// TIA Portal project "Liquid_Level_Control_Factory_IO" (V15)
// Vorlageprojekt für das Buch mit Zielsystem S7-1200

(* hardware
DEVICE "S7-1200-Station_1"  S7-1200 Station
   slot 0: "Baugruppenträger_0"  Rack  V1.0
   slot 1: "Liquid_Level_PLC"  CPU 1211C DC/DC/DC  6ES7 211-1AE40-0XB0  V4.1
DEVICE "Liquid_Level_HMI"  KTP900 Basic PN
   slot 0: "Liquid_Level_HMI"  KTP900 Basic PN  6AV2 123-2JB03-0AX0  15.0.0.0
   slot 1: "HMI_RT_1"  KTP900 Basic PN  6AV2 123-2JB03-0AX0  15.0.0.0
   slot 5: "Liquid_Level_HMI.IE_CP_1"  PROFINET Interface  15.0.0.0
      slot 1: "PROFINET Interface_1"  PROFINET Interface
         slot 1: "Port_1"  Port
*)

// ===== PLC "Liquid_Level_PLC"  CPU 1211C DC/DC/DC =====

VAR_GLOBAL   // PLC tag table "Standard-Variablentabelle"
   "SETPOINT_BUFF" AT %MD100 : DWord;
   "LEVEL_METER_BUFF" AT %MD108 : Real;
   "Discharge_Valve_Buff" AT %MD116 : Real;
END_VAR

VAR_GLOBAL   // PLC tag table "Actuators"
   "START_LGT" AT %Q0.0 : Bool;
   "RESET_LGT" AT %Q0.1 : Bool;
   "STOP_LGT" AT %Q0.2 : Bool;
   "FILL_VALVE" AT %QW30 : Int;
   "DISCHARGE_VALVE" AT %QW32 : Int;
   "WARNING_LGT" AT %Q0.3 : Bool;
   "SIREN" AT %Q0.4 : Bool;
END_VAR

VAR_GLOBAL   // PLC tag table "Sensors"
   "LEVEL_METER" AT %IW30 : Int;
   "FLOW_METER" AT %IW32 : Int;
   "SETPOINT" AT %IW34 : Int;
END_VAR

VAR_GLOBAL   // PLC tag table "Buttons"
   "START_BTN" AT %I0.0 : Bool;
   "RESET_BTN" AT %I0.1 : Bool;
   "STOP_BTN" AT %I0.2 : Bool;
END_VAR

VAR_GLOBAL   // PLC tag table "Display"
   "SP" AT %QW34 : Int;
   "PV" AT %QW36 : Int;
END_VAR

DATA_BLOCK "TANK_CTRL_DB_1"   // DB1
{ S7_Optimized_Access := 'TRUE' }
VERSION : 0.1
   VAR
      PV : Int;
      SP : Int;
      Tank_Lvl : Int;
      Fill_Valve_Pos : Real;
      Valve_Animation : Bool;
      Discharge_Valve : Real;
      Discharge_Animation : Bool;
      In_Error : Int;
      Out_Error : Int;
      Sensor_Error : Int;
      SP_Error : Int;
      Discharge_Error : Int;
      PID_Auto_Bit : Bool;
      PID_Calc_Bit : Bool;
      PID_Mode : Struct
         Enable : Int := 3;
         Disable : Int := 0;
      END_STRUCT;
      PID_Parameters : Struct
         Kp : Real;
         Ti : Real;
         Td : Real;
      END_STRUCT;
      Tuning_Parameters : Struct
         Kp : Real := 2.5;
         Ti : Real := 0.0;
         Td : Real := 0.0;
         Kp_D : Real := 2.5;
         Ti_D : Real := 10.0;
         Td_D : Real := 0.0;
      END_STRUCT;
   END_VAR
   VAR RETAIN
      Calc_Parameters : Struct
         Kp : Real := 2.0;
         Ti : Real := 1.7655;
         Td : Real := 0.0;
      END_STRUCT;
   END_VAR
BEGIN
END_DATA_BLOCK

FUNCTION "Tank_Ctrl" : Void   // FC1, LAD
{ S7_Optimized_Access := 'TRUE' }
VERSION : 0.1
BEGIN

REGION Network 1: SCALE SP
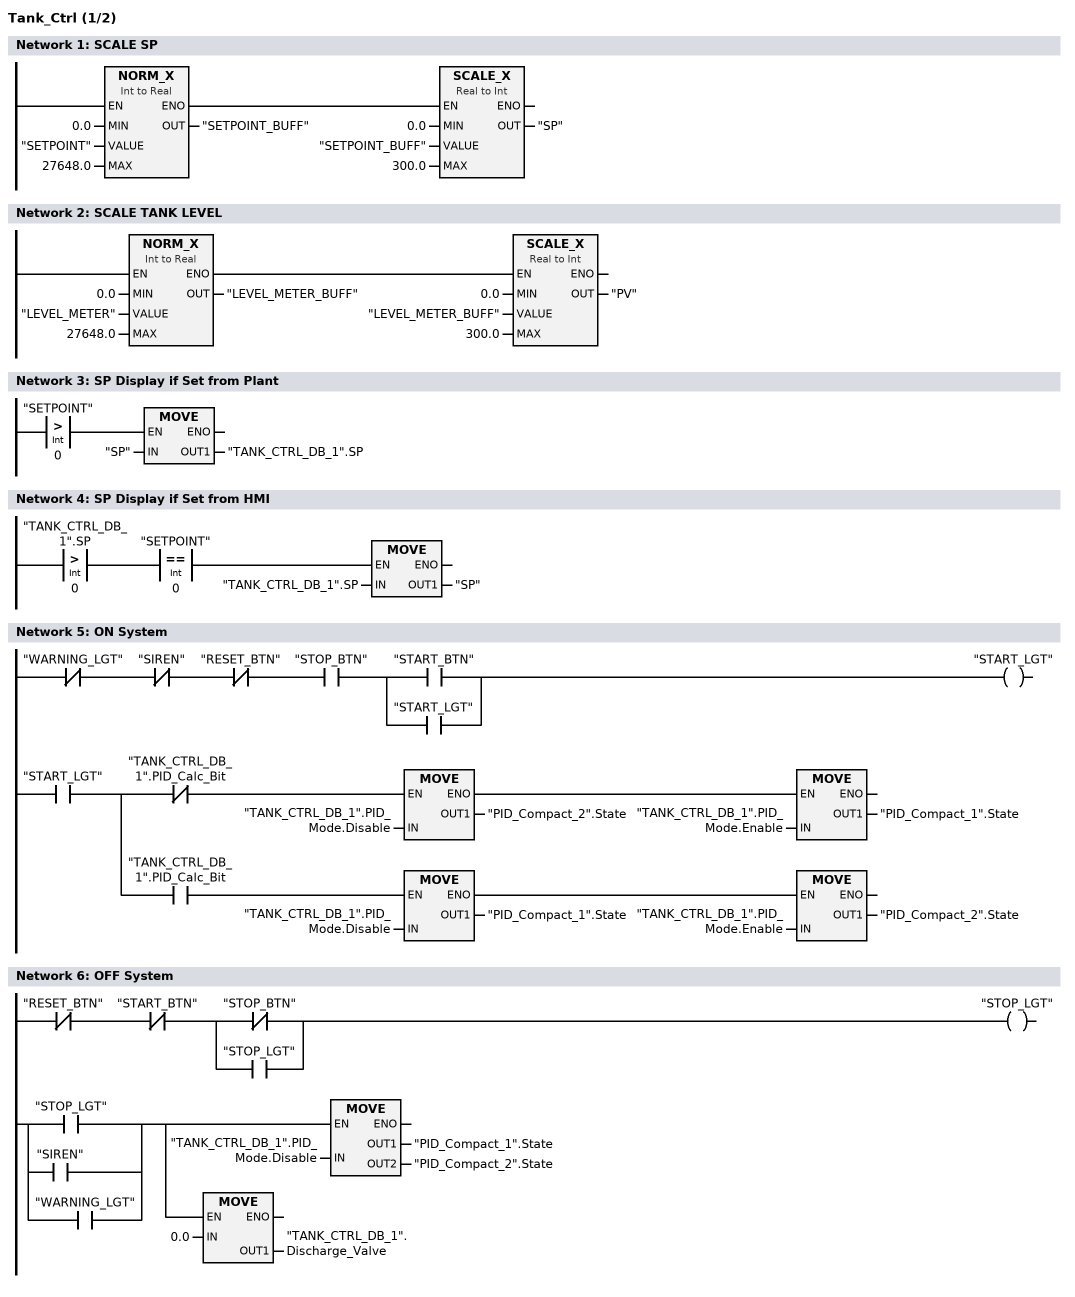
   RUNG wire#powerrail
      { S7_Templates := "[SrcType := Int, DestType := Real]" } Normalize(min := 0.0, value := "SETPOINT", max := 27648.0, out => "SETPOINT_BUFF")
      { S7_Templates := "[SrcType := Real, DestType := Int]" } Scale(min := 0.0, value := "SETPOINT_BUFF", max := 300.0, out => "SP")
   END_RUNG
   // the same network as SCL:
   "SETPOINT_BUFF" := NORM_X(MIN := 0.0, VALUE := "SETPOINT", MAX := 27648.0);
   "SP" := SCALE_X(MIN := 0.0, VALUE := "SETPOINT_BUFF", MAX := 300.0);
END_REGION

REGION Network 2: SCALE TANK LEVEL
   RUNG wire#powerrail
      { S7_Templates := "[SrcType := Int, DestType := Real]" } Normalize(min := 0.0, value := "LEVEL_METER", max := 27648.0, out => "LEVEL_METER_BUFF")
      { S7_Templates := "[SrcType := Real, DestType := Int]" } Scale(min := 0.0, value := "LEVEL_METER_BUFF", max := 300.0, out => "PV")
   END_RUNG
   // the same network as SCL:
   "LEVEL_METER_BUFF" := NORM_X(MIN := 0.0, VALUE := "LEVEL_METER", MAX := 27648.0);
   "PV" := SCALE_X(MIN := 0.0, VALUE := "LEVEL_METER_BUFF", MAX := 300.0);
END_REGION

REGION Network 3: SP Display if Set from Plant
   RUNG wire#powerrail
      { S7_Templates := "SrcType := Int" } GT_Contact(in1 := "SETPOINT", in2 := 0)
      Move(in := "SP", out1 => "TANK_CTRL_DB_1".SP)
   END_RUNG
   // the same network as SCL:
   IF "SETPOINT" > 0 THEN "TANK_CTRL_DB_1".SP := "SP"; END_IF;
END_REGION

REGION Network 4: SP Display if Set from HMI
   RUNG wire#powerrail
      { S7_Templates := "SrcType := Int" } GT_Contact(in1 := "TANK_CTRL_DB_1".SP, in2 := 0)
      { S7_Templates := "SrcType := Int" } EQ_Contact(in1 := "SETPOINT", in2 := 0)
      Move(in := "TANK_CTRL_DB_1".SP, out1 => "SP")
   END_RUNG
   // the same network as SCL:
   IF ("TANK_CTRL_DB_1".SP > 0) AND ("SETPOINT" = 0) THEN "SP" := "TANK_CTRL_DB_1".SP; END_IF;
END_REGION

REGION Network 5: ON System
   RUNG wire#powerrail
      I_Contact( "WARNING_LGT" )
      I_Contact( "SIREN" )
      I_Contact( "RESET_BTN" )
      Contact( "STOP_BTN" )
      wire#w1
      Contact( "START_BTN" )
      wire#w2
      Coil( "START_LGT" )
   END_RUNG
   RUNG wire#w1
      Contact( "START_LGT" )
   END_RUNG wire#w2
   RUNG wire#powerrail
      Contact( "START_LGT" )
      wire#w3
      I_Contact( "TANK_CTRL_DB_1".PID_Calc_Bit )
      Move(in := "TANK_CTRL_DB_1".PID_Mode.Disable, out1 => "PID_Compact_2".State)
      Move(in := "TANK_CTRL_DB_1".PID_Mode.Enable, out1 => "PID_Compact_1".State)
   END_RUNG
   RUNG wire#w3
      Contact( "TANK_CTRL_DB_1".PID_Calc_Bit )
      Move(in := "TANK_CTRL_DB_1".PID_Mode.Disable, out1 => "PID_Compact_1".State)
      Move(in := "TANK_CTRL_DB_1".PID_Mode.Enable, out1 => "PID_Compact_2".State)
   END_RUNG
   // the same network as SCL:
   "START_LGT" := NOT "WARNING_LGT" AND NOT "SIREN" AND NOT "RESET_BTN" AND "STOP_BTN" AND ("START_BTN" OR "START_LGT");
   IF "START_LGT" AND NOT "TANK_CTRL_DB_1".PID_Calc_Bit THEN
       "PID_Compact_2".State := "TANK_CTRL_DB_1".PID_Mode.Disable;
       "PID_Compact_1".State := "TANK_CTRL_DB_1".PID_Mode.Enable;
   END_IF;
   IF "START_LGT" AND "TANK_CTRL_DB_1".PID_Calc_Bit THEN
       "PID_Compact_1".State := "TANK_CTRL_DB_1".PID_Mode.Disable;
       "PID_Compact_2".State := "TANK_CTRL_DB_1".PID_Mode.Enable;
   END_IF;
END_REGION

REGION Network 6: OFF System
   RUNG wire#powerrail
      I_Contact( "RESET_BTN" )
      I_Contact( "START_BTN" )
      wire#w1
      I_Contact( "STOP_BTN" )
      wire#w2
      Coil( "STOP_LGT" )
   END_RUNG
   RUNG wire#w1
      Contact( "STOP_LGT" )
   END_RUNG wire#w2
   RUNG wire#powerrail
      Contact( "STOP_LGT" )
      wire#w3
      Move(in := "TANK_CTRL_DB_1".PID_Mode.Disable, out1 => "PID_Compact_1".State, out2 => "PID_Compact_2".State)
   END_RUNG
   RUNG wire#powerrail
      Contact( "SIREN" )
   END_RUNG wire#w3
   RUNG wire#powerrail
      Contact( "WARNING_LGT" )
   END_RUNG wire#w3
   RUNG wire#w3
      Move(in := 0.0, out1 => "TANK_CTRL_DB_1".Discharge_Valve)
   END_RUNG
   // the same network as SCL:
   "STOP_LGT" := NOT "RESET_BTN" AND NOT "START_BTN" AND (NOT "STOP_BTN" OR "STOP_LGT");
   IF "STOP_LGT" OR "SIREN" OR "WARNING_LGT" THEN
       "PID_Compact_1".State := "TANK_CTRL_DB_1".PID_Mode.Disable;
       "PID_Compact_2".State := "TANK_CTRL_DB_1".PID_Mode.Disable;
       "TANK_CTRL_DB_1".Discharge_Valve := 0.0;
   END_IF;
END_REGION

REGION Network 7: RESET System
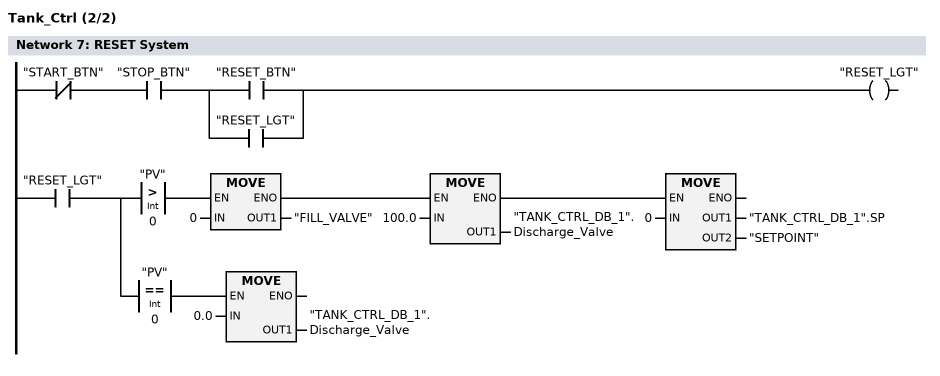
   RUNG wire#powerrail
      I_Contact( "START_BTN" )
      Contact( "STOP_BTN" )
      wire#w1
      Contact( "RESET_BTN" )
      wire#w2
      Coil( "RESET_LGT" )
   END_RUNG
   RUNG wire#w1
      Contact( "RESET_LGT" )
   END_RUNG wire#w2
   RUNG wire#powerrail
      Contact( "RESET_LGT" )
      wire#w3
      { S7_Templates := "SrcType := Int" } GT_Contact(in1 := "PV", in2 := 0)
      Move(in := 0, out1 => "FILL_VALVE")
      Move(in := 100.0, out1 => "TANK_CTRL_DB_1".Discharge_Valve)
      Move(in := 0, out1 => "TANK_CTRL_DB_1".SP, out2 => "SETPOINT")
   END_RUNG
   RUNG wire#w3
      { S7_Templates := "SrcType := Int" } EQ_Contact(in1 := "PV", in2 := 0)
      Move(in := 0.0, out1 => "TANK_CTRL_DB_1".Discharge_Valve)
   END_RUNG
   // the same network as SCL:
   "RESET_LGT" := NOT "START_BTN" AND "STOP_BTN" AND ("RESET_BTN" OR "RESET_LGT");
   IF "RESET_LGT" AND ("PV" > 0) THEN
       "FILL_VALVE" := 0;
       "TANK_CTRL_DB_1".Discharge_Valve := 100.0;
       "TANK_CTRL_DB_1".SP := 0;
       "SETPOINT" := 0;
   END_IF;
   IF "RESET_LGT" AND ("PV" = 0) THEN "TANK_CTRL_DB_1".Discharge_Valve := 0.0; END_IF;
END_REGION
END_FUNCTION

FUNCTION "HMI_Ctrl" : Void   // FC2, LAD
{ S7_Optimized_Access := 'TRUE' }
VERSION : 0.1
   VAR_TEMP   // added for the SCL form of the ladder/FBD networks
      _w1 : Bool;
      _w2 : Bool;
   END_VAR
BEGIN

REGION Network 1: PV and Tank Level
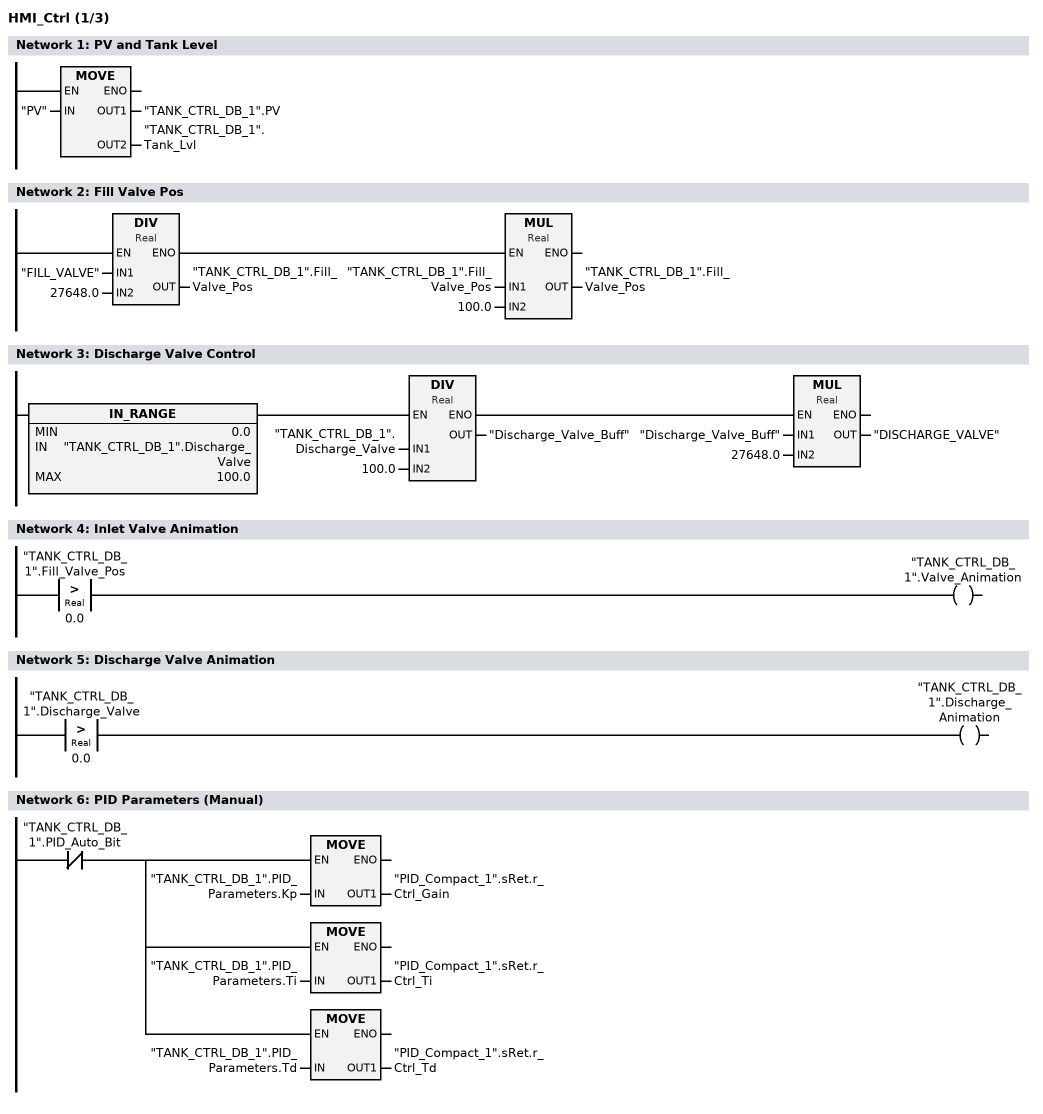
   RUNG wire#powerrail
      Move(in := "PV", out1 => "TANK_CTRL_DB_1".PV, out2 => "TANK_CTRL_DB_1".Tank_Lvl)
   END_RUNG
   // the same network as SCL:
   "TANK_CTRL_DB_1".PV := "PV";
   "TANK_CTRL_DB_1".Tank_Lvl := "PV";
END_REGION

REGION Network 2: Fill Valve Pos
   RUNG wire#powerrail
      { S7_Templates := "SrcType := Real" } Div(in1 := "FILL_VALVE", in2 := 27648.0, out => "TANK_CTRL_DB_1".Fill_Valve_Pos)
      { S7_Templates := "SrcType := Real" } Mul(in1 := "TANK_CTRL_DB_1".Fill_Valve_Pos, in2 := 100.0, out => "TANK_CTRL_DB_1".Fill_Valve_Pos)
   END_RUNG
   // the same network as SCL:
   "TANK_CTRL_DB_1".Fill_Valve_Pos := "FILL_VALVE" / 27648.0;
   "TANK_CTRL_DB_1".Fill_Valve_Pos := "TANK_CTRL_DB_1".Fill_Valve_Pos * 100.0;
END_REGION

REGION Network 3: Discharge Valve Control
   RUNG wire#powerrail
      { S7_Templates := "SrcType := Real" } InRange(min := 0.0, in := "TANK_CTRL_DB_1".Discharge_Valve, max := 100.0)
      { S7_Templates := "SrcType := Real" } Div(in1 := "TANK_CTRL_DB_1".Discharge_Valve, in2 := 100.0, out => "Discharge_Valve_Buff")
      { S7_Templates := "SrcType := Real" } Mul(in1 := "Discharge_Valve_Buff", in2 := 27648.0, out => "DISCHARGE_VALVE")
   END_RUNG
   // the same network as SCL:
   IF (0.0 <= "TANK_CTRL_DB_1".Discharge_Valve) AND ("TANK_CTRL_DB_1".Discharge_Valve <= 100.0) THEN
       "Discharge_Valve_Buff" := "TANK_CTRL_DB_1".Discharge_Valve / 100.0;
       "DISCHARGE_VALVE" := "Discharge_Valve_Buff" * 27648.0;
   END_IF;
END_REGION

REGION Network 4: Inlet Valve Animation
   RUNG wire#powerrail
      { S7_Templates := "SrcType := Real" } GT_Contact(in1 := "TANK_CTRL_DB_1".Fill_Valve_Pos, in2 := 0.0)
      Coil( "TANK_CTRL_DB_1".Valve_Animation )
   END_RUNG
   // the same network as SCL:
   "TANK_CTRL_DB_1".Valve_Animation := "TANK_CTRL_DB_1".Fill_Valve_Pos > 0.0;
END_REGION

REGION Network 5: Discharge Valve Animation
   RUNG wire#powerrail
      { S7_Templates := "SrcType := Real" } GT_Contact(in1 := "TANK_CTRL_DB_1".Discharge_Valve, in2 := 0.0)
      Coil( "TANK_CTRL_DB_1".Discharge_Animation )
   END_RUNG
   // the same network as SCL:
   "TANK_CTRL_DB_1".Discharge_Animation := "TANK_CTRL_DB_1".Discharge_Valve > 0.0;
END_REGION

REGION Network 6: PID Parameters (Manual)
   RUNG wire#powerrail
      I_Contact( "TANK_CTRL_DB_1".PID_Auto_Bit )
      wire#w1
      Move(in := "TANK_CTRL_DB_1".PID_Parameters.Kp, out1 => "PID_Compact_1".sRet.r_Ctrl_Gain)
   END_RUNG
   RUNG wire#w1
      Move(in := "TANK_CTRL_DB_1".PID_Parameters.Ti, out1 => "PID_Compact_1".sRet.r_Ctrl_Ti)
   END_RUNG
   RUNG wire#w1
      Move(in := "TANK_CTRL_DB_1".PID_Parameters.Td, out1 => "PID_Compact_1".sRet.r_Ctrl_Td)
   END_RUNG
   // the same network as SCL:
   IF NOT "TANK_CTRL_DB_1".PID_Auto_Bit THEN
       "PID_Compact_1".sRet.r_Ctrl_Gain := "TANK_CTRL_DB_1".PID_Parameters.Kp;
       "PID_Compact_1".sRet.r_Ctrl_Ti := "TANK_CTRL_DB_1".PID_Parameters.Ti;
       "PID_Compact_1".sRet.r_Ctrl_Td := "TANK_CTRL_DB_1".PID_Parameters.Td;
   END_IF;
END_REGION

REGION Network 7: PID Parameters (Automatic, Trial)
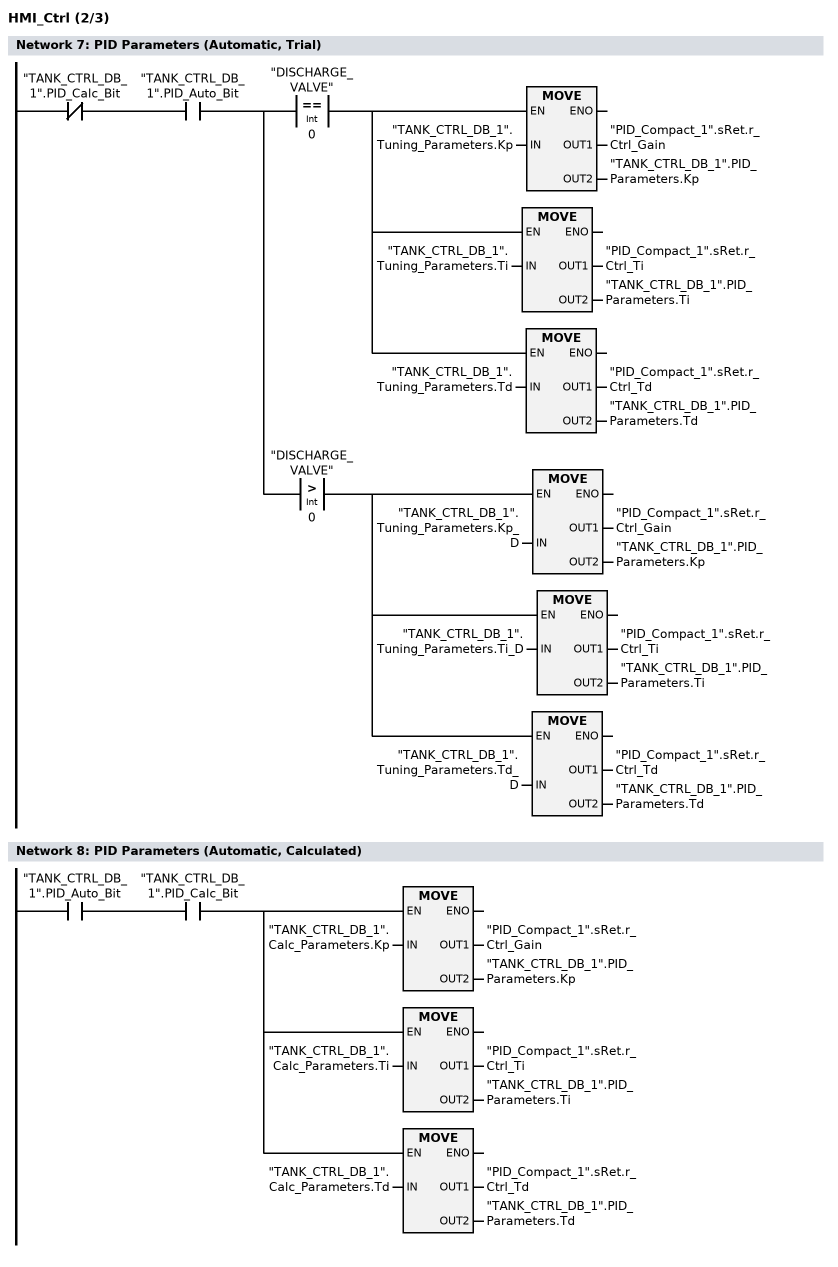
   RUNG wire#powerrail
      I_Contact( "TANK_CTRL_DB_1".PID_Calc_Bit )
      Contact( "TANK_CTRL_DB_1".PID_Auto_Bit )
      wire#w1
      { S7_Templates := "SrcType := Int" } EQ_Contact(in1 := "DISCHARGE_VALVE", in2 := 0)
      wire#w2
      Move(in := "TANK_CTRL_DB_1".Tuning_Parameters.Kp, out1 => "PID_Compact_1".sRet.r_Ctrl_Gain, out2 => "TANK_CTRL_DB_1".PID_Parameters.Kp)
   END_RUNG
   RUNG wire#w2
      Move(in := "TANK_CTRL_DB_1".Tuning_Parameters.Ti, out1 => "PID_Compact_1".sRet.r_Ctrl_Ti, out2 => "TANK_CTRL_DB_1".PID_Parameters.Ti)
   END_RUNG
   RUNG wire#w2
      Move(in := "TANK_CTRL_DB_1".Tuning_Parameters.Td, out1 => "PID_Compact_1".sRet.r_Ctrl_Td, out2 => "TANK_CTRL_DB_1".PID_Parameters.Td)
   END_RUNG
   RUNG wire#w1
      { S7_Templates := "SrcType := Int" } GT_Contact(in1 := "DISCHARGE_VALVE", in2 := 0)
      wire#w3
      Move(in := "TANK_CTRL_DB_1".Tuning_Parameters.Kp_D, out1 => "PID_Compact_1".sRet.r_Ctrl_Gain, out2 => "TANK_CTRL_DB_1".PID_Parameters.Kp)
   END_RUNG
   RUNG wire#w3
      Move(in := "TANK_CTRL_DB_1".Tuning_Parameters.Ti_D, out1 => "PID_Compact_1".sRet.r_Ctrl_Ti, out2 => "TANK_CTRL_DB_1".PID_Parameters.Ti)
   END_RUNG
   RUNG wire#w3
      Move(in := "TANK_CTRL_DB_1".Tuning_Parameters.Td_D, out1 => "PID_Compact_1".sRet.r_Ctrl_Td, out2 => "TANK_CTRL_DB_1".PID_Parameters.Td)
   END_RUNG
   // the same network as SCL:
   #_w1 := NOT "TANK_CTRL_DB_1".PID_Calc_Bit AND "TANK_CTRL_DB_1".PID_Auto_Bit;
   IF #_w1 AND ("DISCHARGE_VALVE" = 0) THEN
       "PID_Compact_1".sRet.r_Ctrl_Gain := "TANK_CTRL_DB_1".Tuning_Parameters.Kp;
       "TANK_CTRL_DB_1".PID_Parameters.Kp := "TANK_CTRL_DB_1".Tuning_Parameters.Kp;
       "PID_Compact_1".sRet.r_Ctrl_Ti := "TANK_CTRL_DB_1".Tuning_Parameters.Ti;
       "TANK_CTRL_DB_1".PID_Parameters.Ti := "TANK_CTRL_DB_1".Tuning_Parameters.Ti;
       "PID_Compact_1".sRet.r_Ctrl_Td := "TANK_CTRL_DB_1".Tuning_Parameters.Td;
       "TANK_CTRL_DB_1".PID_Parameters.Td := "TANK_CTRL_DB_1".Tuning_Parameters.Td;
   END_IF;
   IF #_w1 AND ("DISCHARGE_VALVE" > 0) THEN
       "PID_Compact_1".sRet.r_Ctrl_Gain := "TANK_CTRL_DB_1".Tuning_Parameters.Kp_D;
       "TANK_CTRL_DB_1".PID_Parameters.Kp := "TANK_CTRL_DB_1".Tuning_Parameters.Kp_D;
       "PID_Compact_1".sRet.r_Ctrl_Ti := "TANK_CTRL_DB_1".Tuning_Parameters.Ti_D;
       "TANK_CTRL_DB_1".PID_Parameters.Ti := "TANK_CTRL_DB_1".Tuning_Parameters.Ti_D;
       "PID_Compact_1".sRet.r_Ctrl_Td := "TANK_CTRL_DB_1".Tuning_Parameters.Td_D;
       "TANK_CTRL_DB_1".PID_Parameters.Td := "TANK_CTRL_DB_1".Tuning_Parameters.Td_D;
   END_IF;
END_REGION

REGION Network 8: PID Parameters (Automatic, Calculated)
   RUNG wire#powerrail
      Contact( "TANK_CTRL_DB_1".PID_Auto_Bit )
      Contact( "TANK_CTRL_DB_1".PID_Calc_Bit )
      wire#w1
      Move(in := "TANK_CTRL_DB_1".Calc_Parameters.Kp, out1 => "PID_Compact_1".sRet.r_Ctrl_Gain, out2 => "TANK_CTRL_DB_1".PID_Parameters.Kp)
   END_RUNG
   RUNG wire#w1
      Move(in := "TANK_CTRL_DB_1".Calc_Parameters.Ti, out1 => "PID_Compact_1".sRet.r_Ctrl_Ti, out2 => "TANK_CTRL_DB_1".PID_Parameters.Ti)
   END_RUNG
   RUNG wire#w1
      Move(in := "TANK_CTRL_DB_1".Calc_Parameters.Td, out1 => "PID_Compact_1".sRet.r_Ctrl_Td, out2 => "TANK_CTRL_DB_1".PID_Parameters.Td)
   END_RUNG
   // the same network as SCL:
   IF "TANK_CTRL_DB_1".PID_Auto_Bit AND "TANK_CTRL_DB_1".PID_Calc_Bit THEN
       "PID_Compact_1".sRet.r_Ctrl_Gain := "TANK_CTRL_DB_1".Calc_Parameters.Kp;
       "TANK_CTRL_DB_1".PID_Parameters.Kp := "TANK_CTRL_DB_1".Calc_Parameters.Kp;
       "PID_Compact_1".sRet.r_Ctrl_Ti := "TANK_CTRL_DB_1".Calc_Parameters.Ti;
       "TANK_CTRL_DB_1".PID_Parameters.Ti := "TANK_CTRL_DB_1".Calc_Parameters.Ti;
       "PID_Compact_1".sRet.r_Ctrl_Td := "TANK_CTRL_DB_1".Calc_Parameters.Td;
       "TANK_CTRL_DB_1".PID_Parameters.Td := "TANK_CTRL_DB_1".Calc_Parameters.Td;
   END_IF;
END_REGION

REGION Network 9: Warnings
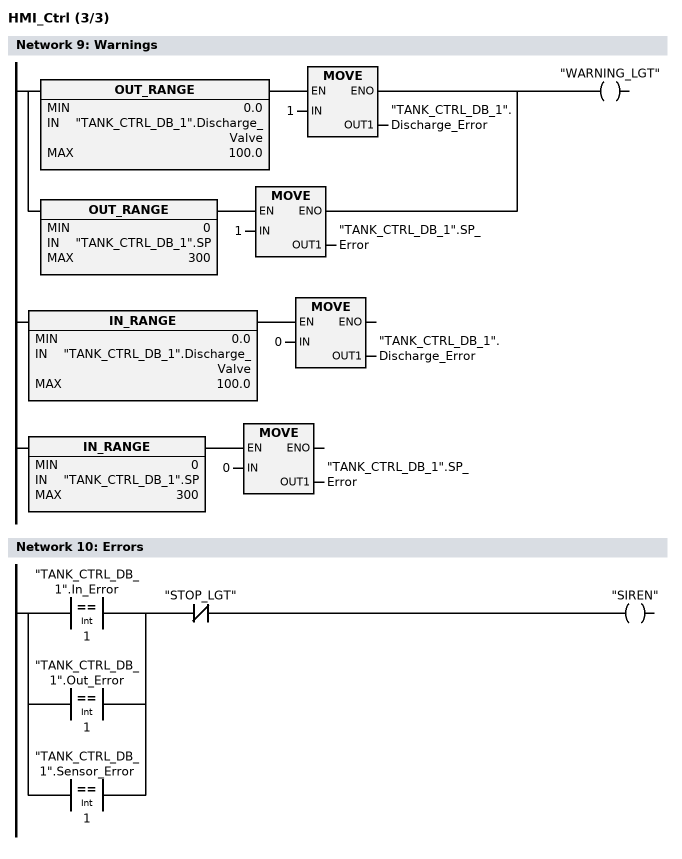
   #_w1 := ("TANK_CTRL_DB_1".Discharge_Valve < 0.0) OR ("TANK_CTRL_DB_1".Discharge_Valve > 100.0);
   IF #_w1 THEN "TANK_CTRL_DB_1".Discharge_Error := 1; END_IF;
   #_w2 := ("TANK_CTRL_DB_1".SP < 0) OR ("TANK_CTRL_DB_1".SP > 300);
   IF #_w2 THEN "TANK_CTRL_DB_1".SP_Error := 1; END_IF;
   "WARNING_LGT" := #_w1 OR #_w2;
   IF (0.0 <= "TANK_CTRL_DB_1".Discharge_Valve) AND ("TANK_CTRL_DB_1".Discharge_Valve <= 100.0) THEN
       "TANK_CTRL_DB_1".Discharge_Error := 0;
   END_IF;
   IF (0 <= "TANK_CTRL_DB_1".SP) AND ("TANK_CTRL_DB_1".SP <= 300) THEN
       "TANK_CTRL_DB_1".SP_Error := 0;
   END_IF;
END_REGION

REGION Network 10: Errors
   RUNG wire#powerrail
      { S7_Templates := "SrcType := Int" } EQ_Contact(in1 := "TANK_CTRL_DB_1".In_Error, in2 := 1)
      wire#w1
      I_Contact( "STOP_LGT" )
      Coil( "SIREN" )
   END_RUNG
   RUNG wire#powerrail
      { S7_Templates := "SrcType := Int" } EQ_Contact(in1 := "TANK_CTRL_DB_1".Out_Error, in2 := 1)
   END_RUNG wire#w1
   RUNG wire#powerrail
      { S7_Templates := "SrcType := Int" } EQ_Contact(in1 := "TANK_CTRL_DB_1".Sensor_Error, in2 := 1)
   END_RUNG wire#w1
   // the same network as SCL:
   "SIREN" := (("TANK_CTRL_DB_1".In_Error = 1) OR ("TANK_CTRL_DB_1".Out_Error = 1) OR ("TANK_CTRL_DB_1".Sensor_Error = 1)) AND NOT "STOP_LGT";
END_REGION
END_FUNCTION

FUNCTION "MHJ-PLC-Lab-Function-S71200" : Void   // FC9000, SCL
{ S7_Optimized_Access := 'TRUE' }
VERSION : 0.1
   VAR_TEMP
      rdTimeReturn : Int;
      outputTime : DTL;
      SyncVal : Byte;
      forVal : Int;
      forVal_2 : Int;
      Value : Byte;
   END_VAR
   VAR CONSTANT
      CompVal : Byte := 16#34;
      Value_01 : Byte := 16#11;
      Value_01_DW : DWord := 16#A165_D992;
      Value_02_DW : DWord := 16#58BE_4401;
   END_VAR
BEGIN

   #Value:=PEEK(area := 16#82,
        dbNumber := 0,
        byteOffset := 511);
   #Value := #Value + 1;

   POKE(area := 16#82,
        dbNumber := 0,
        byteOffset := 511,
        value := #Value);

   POKE(area:=16#81,
        dbNumber:=0,
        byteOffset:=1016,
        value:=#Value_01_DW);
   POKE(area := 16#81,
        dbNumber := 0,
        byteOffset := 1020,
        value := #Value_02_DW);

   POKE(area := 16#81,
        dbNumber := 0,
        byteOffset := 511,
        value := B#16#00);

   FOR #forVal := 0 TO 120 DO
       FOR #forVal_2:=0 TO 10 DO
           #rdTimeReturn:=RD_SYS_T(#outputTime);
           #rdTimeReturn := WR_SYS_T(#outputTime);
           #rdTimeReturn := RD_SYS_T(#outputTime);
           #rdTimeReturn := WR_SYS_T(#outputTime);
       END_FOR;
       #SyncVal:= PEEK(area := 16#81,
                      dbNumber := 0,
                      byteOffset := 511);
       IF #SyncVal = #CompVal THEN
          GOTO M_1;
       END_IF;
   END_FOR;
   RETURN;

   M_1:
   POKE(area := 16#81,
        dbNumber := 0,
        byteOffset := 511,
        value := B#16#0);
END_FUNCTION

ORGANIZATION_BLOCK "Main"   // OB1, FBD, ProgramCycle
TITLE = "Main Program Sweep (Cycle)"
{ S7_Optimized_Access := 'TRUE' }
VERSION : 0.1
   VAR_INPUT
      Initial_Call : Bool;   // Initial call of this OB
      Remanence : Bool;   // =True, if remanent data are available
   END_VAR
BEGIN

REGION Network 1: Konnektierungsbaustein für PLC-Lab / TIA PORTAL CONNECTION TO FACTORY IO
   // Im Netzwerk 1 wird der Konnektierungsbaustein für PLC-Lab aufgerufen.
   // Dieser Aufruf darf nicht entfernt werden!
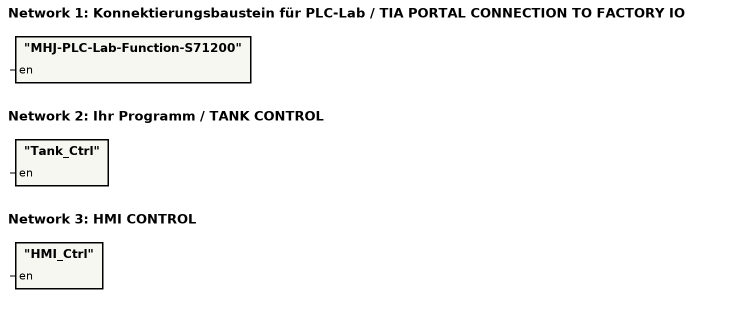
   "MHJ-PLC-Lab-Function-S71200"();
END_REGION

REGION Network 2: Ihr Programm / TANK CONTROL
   // Schreiben Sie ab Netzwerk 2 Ihr Programm
   "Tank_Ctrl"();
END_REGION

REGION Network 3: HMI CONTROL
   "HMI_Ctrl"();
END_REGION
END_ORGANIZATION_BLOCK

ORGANIZATION_BLOCK "PID_Controller"   // OB30, LAD, CyclicInterrupt
TITLE = Inlet Valve Controller
{ S7_Optimized_Access := 'TRUE' }
VERSION : 0.1
   VAR_INPUT
      Initial_Call : Bool;   // Initial call of this OB
      Event_Count : Int;   // Events discarded
   END_VAR
BEGIN

REGION Network 1: PID Control (Fine Tuned)
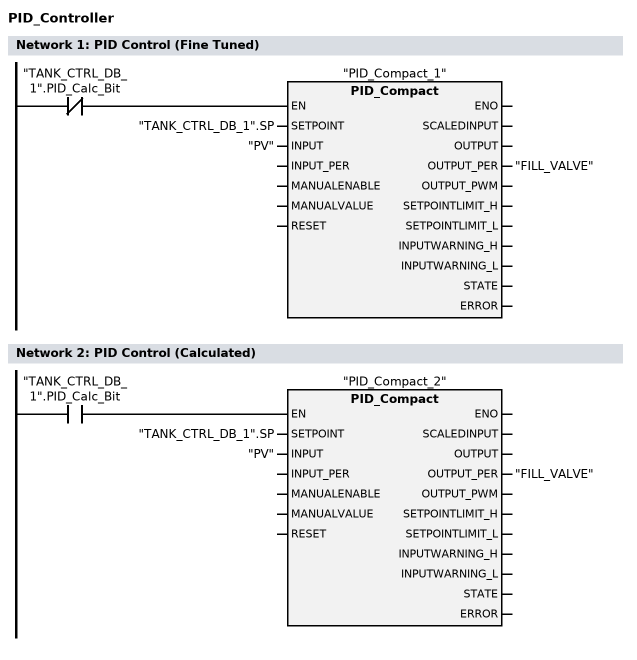
   IF NOT "TANK_CTRL_DB_1".PID_Calc_Bit THEN
       "PID_Compact_1"(Setpoint := "TANK_CTRL_DB_1".SP, Input := "PV", Output_PER => "FILL_VALVE");   // PID_Compact
   END_IF;
END_REGION

REGION Network 2: PID Control (Calculated)
   IF "TANK_CTRL_DB_1".PID_Calc_Bit THEN
       "PID_Compact_2"(Setpoint := "TANK_CTRL_DB_1".SP, Input := "PV", Output_PER => "FILL_VALVE");   // PID_Compact
   END_IF;
END_REGION
END_ORGANIZATION_BLOCK

(* ===== HMI "HMI_RT_1" =====
system functions are stored by id; their names below are inferred from use
connection "HMI_Connection_1": ETHERNET, SMART_S7_1200_OMS

HMI tags "Default tag table"
   "Tag_ScreenNumber" : UInt, internal
   "TANK_CTRL_DB_1_In_Error" : Int = PLC TANK_CTRL_DB_1.In_Error, 1 s
   "TANK_CTRL_DB_1_Out_Error" : Int = PLC TANK_CTRL_DB_1.Out_Error, 1 s
   "TANK_CTRL_DB_1_Sensor_Error" : Int = PLC TANK_CTRL_DB_1.Sensor_Error, 1 s
   "TANK_CTRL_DB_1_SP" : Int = PLC TANK_CTRL_DB_1.SP, 1 s
   "TANK_CTRL_DB_1_PV" : Int = PLC TANK_CTRL_DB_1.PV, 1 s
   "TANK_CTRL_DB_1_Fill_Valve_Pos" : Real = PLC TANK_CTRL_DB_1.Fill_Valve_Pos, 1 s
   "TANK_CTRL_DB_1_Tank_Lvl" : Int = PLC TANK_CTRL_DB_1.Tank_Lvl, 1 s
   "TANK_CTRL_DB_1_Valve_Animation" : Bool = PLC TANK_CTRL_DB_1.Valve_Animation, 1 s
   "TANK_CTRL_DB_1_Discharge_Animation" : Bool = PLC TANK_CTRL_DB_1.Discharge_Animation, 1 s
   "TANK_CTRL_DB_1_PID_Calc_Bit" : Bool = PLC TANK_CTRL_DB_1.PID_Calc_Bit, 1 s
   "TANK_CTRL_DB_1_PID_Auto_Bit" : Bool = PLC TANK_CTRL_DB_1.PID_Auto_Bit, 1 s
   "START_BTN" : Bool = PLC START_BTN AT %I0.0, 1 s
   "STOP_BTN" : Bool = PLC STOP_BTN AT %I0.2, 1 s
   "RESET_BTN" : Bool = PLC RESET_BTN AT %I0.1, 1 s
   "TANK_CTRL_DB_1_Discharge_Valve" : Real = PLC TANK_CTRL_DB_1.Discharge_Valve, 1 s
   "TANK_CTRL_DB_1_PID_Parameters_Kp" : Real = PLC TANK_CTRL_DB_1.PID_Parameters.Kp, 1 s
   "TANK_CTRL_DB_1_PID_Parameters_Ti" : Real = PLC TANK_CTRL_DB_1.PID_Parameters.Ti, 1 s
   "TANK_CTRL_DB_1_PID_Parameters_Td" : Real = PLC TANK_CTRL_DB_1.PID_Parameters.Td, 1 s

Template "Template_1" 800x480
   Button "Exit" at 722,440 size 55x39; TextOff 'Exit'; PictureOff "ExitRuntime_KTP900_Basic_PN_TR"; PictureOn "ExitRuntime_KTP900_Basic_PN_TR"
      on Release: StopRuntime(0)
   Button "Template_Button" at 622,440 size 55x39; TextOff 'Text'
   Button "Template_Button_1" at 522,440 size 55x39; TextOff 'Text'
   Button "Template_Button_2" at 422,440 size 55x39; TextOff 'Text'
   Button "Template_Button_3" at 322,440 size 55x39; TextOff 'Text'
   Button "Template_Button_4" at 222,440 size 55x39; TextOff 'Text'
   Button "Alarms" at 122,440 size 55x39; TextOff 'Alarms'; PictureOff "AlarmDisplay_KTP900_Basic_PN_TR"; PictureOn "AlarmDisplay_KTP900_Basic_PN_TR"
      on Release: function_ef3f5d25("Alarm window_Unacknowledged", -1)
   Button "Start screen" at 22,440 size 55x39; TextOff 'Start screen'; PictureOff "NavigateHome_KTP900_Basic_PN_TR"; PictureOn "NavigateHome_KTP900_Basic_PN_TR"
      on Release: ActivateScreen("Master", 0)
   SymbolicIOField "Symbolic_IO_Field_Screen" at 73,7 size 620x26; TextOff '0'; TextOn '1'; TextList "TextList_ScreenNames"
      ProcessValue <- "Tag_ScreenNumber"
      on Change: ActivateScreenByNumber("Tag_ScreenNumber", 0)
   DateTimeField "HmiScreenItemData" at 695,20 size 105x20
   DateTimeField "HmiScreenItemData_1" at 695,0 size 105x20
   GraphicView "Logo" at 0,0 size 71x40; Picture "Logo of HMI_1"

screen "Master" 800x480, template "Template_1"
   on GenerateScreen: SetTag("Tag_ScreenNumber", 1)
   GraphicView "Graphic view_1" at 32,89 size 195x333; Picture "Graphic_1"
   GraphicView "Graphic view_2" at 204,82 size 56x70; Picture "Graphic_2"
      Visibility <- "TANK_CTRL_DB_1_Valve_Animation"
   GraphicView "Graphic view_3" at 204,288 size 56x70; Picture "Graphic_2"
      Visibility <- "TANK_CTRL_DB_1_Discharge_Animation"
   Bar "Bar_1" at 59,115 size 145x228; MinimumValue 0; MaximumValue 300
      ProcessValue <- "TANK_CTRL_DB_1_Tank_Lvl"
   TextField "Text field_1" at 58,58 size 162x27; Text 'VISUALIZATION'
   TextField "Text field_2" at 284,58 size 241x27; Text 'PROCESS INDICATORS'
   TextField "Text field_3" at 585,58 size 172x27; Text 'PID CONTROL'
   TextField "Text field_4" at 285,312 size 241x27; Text 'DISCHARGE CONTROL'
   TextField "Text field_5" at 400,117 size 137x27; Text 'SP'
   TextField "Text field_6" at 399,180 size 137x27; Text 'PV'
   TextField "Text field_7" at 399,244 size 137x27; Text '% INLET'
   TextField "Text field_8" at 370,369 size 166x27; Text '% DISCHARGE'
   Button "Button_1" at 558,325 size 107x44; TextOff 'START'
      on Click: SetBit("START_BTN")
   Button "Button_2" at 673,325 size 104x44; TextOff 'STOP'
      on Click: ResetBit("STOP_BTN")
   Button "Button_3" at 615,375 size 108x45; TextOff 'RESET'
      on Click: SetBit("RESET_BTN")
   Switch "Switch_1" at 555,94 size 116x32; CaptionText 'Switch'; TextOff 'MANUAL'; TextOn 'AUTO'
      ProcessValue <- "TANK_CTRL_DB_1_PID_Auto_Bit"
   Switch "Switch_2" at 676,94 size 107x32; CaptionText 'Switch'; TextOff 'TRIAL'; TextOn 'CALC'
      ProcessValue <- "TANK_CTRL_DB_1_PID_Calc_Bit"
   IOField "I/O field_1" at 310,115 size 96x32; FormatPattern 99999
      ProcessValue <- "TANK_CTRL_DB_1_SP"
   IOField "I/O field_2" at 310,178 size 96x32; FormatPattern 99999
      ProcessValue <- "TANK_CTRL_DB_1_PV"
   IOField "I/O field_3" at 310,242 size 96x32; FormatPattern 99999.99
      ProcessValue <- "TANK_CTRL_DB_1_Fill_Valve_Pos"
   IOField "I/O field_4" at 281,367 size 96x32; FormatPattern s99999
      ProcessValue <- "TANK_CTRL_DB_1_Discharge_Valve"
   IOField "I/O field_5" at 576,142 size 96x32; FormatPattern 999999999.999
      ProcessValue <- "TANK_CTRL_DB_1_PID_Parameters_Kp"
   IOField "I/O field_6" at 576,203 size 96x32; FormatPattern 999999999.999
      ProcessValue <- "TANK_CTRL_DB_1_PID_Parameters_Ti"
   IOField "I/O field_7" at 576,267 size 96x32; FormatPattern 999999999.999
      ProcessValue <- "TANK_CTRL_DB_1_PID_Parameters_Td"
   TextField "Text field_9" at 662,141 size 137x27; Text 'Kp'
   TextField "Text field_10" at 661,204 size 137x27; Text 'Ti'
   TextField "Text field_11" at 661,268 size 137x27; Text 'Td'

screen "Graphs" 800x480, template "Template_1"
   on GenerateScreen: SetTag("Tag_ScreenNumber", 2)
   Button "Back" at 1,41 size 159x47; TextOff 'Back'
      on Release: ActivateScreen("Master", 0)
   TrendView "Trend view_1" at 10,91 size 779x343

screen "Alarms" 800x480, template "Template_1"
   on GenerateScreen: SetTag("Tag_ScreenNumber", 3)
   Button "Back" at 1,41 size 159x47; TextOff 'Back'
      on Release: ActivateScreen("Master", 0)
   AlarmView "Alarm view_1" at 9,91 size 782x289
   Button "Button_2" at 143,396 size 96x32; TextOn 'BROKEN'; TextOff 'INLET'
      on Press: function_b14e0dd5("TANK_CTRL_DB_1_In_Error", 0)
   Button "Button_4" at 351,396 size 96x32; TextOn 'BROKEN'; TextOff 'DISCHARGE'
      on Press: function_b14e0dd5("TANK_CTRL_DB_1_Out_Error", 0)
   Button "Button_6" at 559,396 size 96x32; TextOn 'BROKEN'; TextOff 'SENSOR'
      on Press: function_b14e0dd5("TANK_CTRL_DB_1_Sensor_Error", 0)
*)